PROGRAM brightspace
VAR
	
	TaskMaster: ARRAY[1..2, 1..3] OF INT := [
        0, 0, 1,    // 30 day task
        0, 0, 1     // 10 day task
    ];

	TasksGiven: INT;
	
	
END_VAR

//how many days till certain assignment needs to be done
GVL.MainDueIn := TaskMaster[1, 2] - GVL.Day;

//make task
IF TaskMaster[1, 1] = 0 OR GVL.MainDueIn < 0 AND TaskMaster[1,3] = 1 THEN
	TaskMaster[1, 1] := TasksGiven + 1;
	TaskMaster[1, 2] := GVL.Day + 30;
	TaskMaster[1, 3] := 0;
	GVL.Finished := FALSE;
	TasksGiven := TasksGiven +1;
	GVL.StartPls := TRUE;
END_IF

//arrays and global variables dont mix
IF GVL.Finished = TRUE THEN				//yes im using this if statement as an SR flipflop
	TaskMaster[1, 3] := 1;
END_IF
 
//send signal once to remind the student to pls start doing something
IF GVL.MainDueIn = 30 AND TaskMaster[1,3] = 0 OR GVL.MainDueIn = 20 AND TaskMaster[1,3] = 0 OR GVL.MainDueIn = 10 AND TaskMaster[1,3] = 0 OR GVL.MainDueIn = 1 AND TaskMaster[1,3] = 0 THEN 
	GVL.StartPls := TRUE;
ELSE
	GVL.StartPls := FALSE;		
END_IF

END_PROGRAM

(* stored: Version 1.1.0.1, ProductVersion 3.1.4024.12
   POU brightspace: Id {1627b2b4-c2df-41ad-9fd7-5cb03a7c9461}, SpecialFunc None *)
